// TwinCAT 3 PLC project M1L0_PLC
// ProgramVersion: 3.1.4020.5
// libraries:
//   Tc2_MC2, * (Beckhoff Automation GmbH)
//   Tc2_Standard, * (Beckhoff Automation GmbH)
//   Tc2_System, * (Beckhoff Automation GmbH)
//   Tc2_Utilities, * (Beckhoff Automation GmbH)
//   Tc3_Module, * (Beckhoff Automation GmbH)
//   lcls-twincat-motion,0.0.0,SLAC
// project tree:
//   / PlcTask.TcTTO
//   POUs/ MAIN.TcPOU
// real-time tasks:
//   TASK PlcTask: cycle T#10ms, priority 20, ADS port 350
// motion (NC):
//   TASK NC-Task 1 SAF: cycle T#2ms, priority 4, ADS port 501
//   TASK NC-Task 1 SVB: cycle T#10ms, priority 8, ADS port 511
//   AXIS Axis_Yup (id 1)
//     Dynamic: Acceleration=0.2, Deceleration=0.2, DelayTime=0.008
//     Velo: Maximum=0.45
//     OtherSettings: AllowMotionCmdToSlave=true
//     encoder EncType=1
//       EncPara: ScaleFactorNumerator=1e-006
//     drive DrvType=5
//       DrvPara: Inverse=true
//         Analog: VeloReferenz=0.48828125, ScaleFactorActTorque=0.1
//         TimeComp: TaskDelayCycles=1
//     controller CtrType=2
//       CtrPara: PriorControlFactor=1
//         PosDiffControl: Range=0.5
//         PID: PosKp=20, PosExtKp=5, DeadBandPosition=0.0004
//         Observer: BandWidth=20
//   AXIS Axis_Ydwn (id 2)
//     Dynamic: Acceleration=0.2, Deceleration=0.2, DelayTime=0.008
//     Velo: Maximum=0.45
//     OtherSettings: AllowMotionCmdToSlave=true
//     encoder EncType=1
//       EncPara: ScaleFactorNumerator=1e-006
//     drive DrvType=5
//       DrvPara: Inverse=true
//         Analog: VeloReferenz=0.48828125, ScaleFactorActTorque=0.1
//         TimeComp: TaskDelayCycles=1
//     controller CtrType=2
//       CtrPara: PriorControlFactor=1
//         PosDiffControl: Range=0.5
//         PID: PosKp=20, PosExtKp=5, DeadBandPosition=0.0004
//         Observer: BandWidth=20
//   AXIS Axis_Xup (id 3)
//     Dynamic: Acceleration=2, Deceleration=2, DelayTime=0.008
//     Velo: Maximum=1
//     OtherSettings: AllowMotionCmdToSlave=true
//     encoder EncType=1
//       EncPara: ScaleFactorNumerator=1e-006
//     drive DrvType=5
//       Analog: VeloReferenz=1.220703125, ScaleFactorActTorque=0.1
//       TimeComp: TaskDelayCycles=1
//     controller CtrType=2
//       CtrPara: PriorControlFactor=1
//         PosDiffControl: Range=0.1
//         PID: PosKp=10, PosExtKp=1, DeadBandPosition=0.0004
//         Observer: BandWidth=20
//   AXIS Axis_Xdwn (id 4)
//     Dynamic: Acceleration=2, Deceleration=2, DelayTime=0.008
//     Velo: Maximum=1
//     OtherSettings: AllowMotionCmdToSlave=true
//     encoder EncType=1
//       EncPara: ScaleFactorNumerator=1e-006
//     drive DrvType=5
//       DrvPara: Inverse=true
//         Analog: VeloReferenz=1.220703125, ScaleFactorActTorque=0.1
//         TimeComp: TaskDelayCycles=1
//     controller CtrType=2
//       CtrPara: PriorControlFactor=1
//         PosDiffControl: Range=0.1
//         PID: PosKp=10, PosExtKp=1, DeadBandPosition=0.0004
//         Observer: BandWidth=20
//   AXIS Axis_PitchCoarse (id 5)
//     General: UnitName=urad
//     Dynamic: Acceleration=390, Deceleration=390, DelayTime=0.008
//     Velo: Maximum=760
//     OtherSettings: AllowMotionCmdToSlave=true
//     encoder EncType=1
//       EncPara: ScaleFactorNumerator=0.001949317739
//     drive DrvType=5
//       Analog: VeloReferenz=761.4522417, ScaleFactorActTorque=0.1
//       TimeComp: TaskDelayCycles=1
//     controller CtrType=2
//       CtrPara: PriorControlFactor=1
//         PosDiffControl: Range=150
//         PID: PosKp=10, PosExtKp=1, DeadBandPosition=0.1
//         Observer: BandWidth=20
//   AXIS Axis_Bender (id 6)
//     Dynamic: Acceleration=0.1, Deceleration=0.1, DelayTime=0.008
//     Velo: Maximum=0.19
//     OtherSettings: AllowMotionCmdToSlave=true
//     encoder EncType=1
//       EncPara: ScaleFactorNumerator=1e-006
//     drive DrvType=5
//       Analog: VeloReferenz=0.1953125, ScaleFactorActTorque=0.1
//       TimeComp: TaskDelayCycles=1
//     controller CtrType=2
//       CtrPara: PriorControlFactor=1
//         PosDiffControl: Range=0.005
//         PID: PosKp=10, PosExtKp=1, DeadBandPosition=4e-005
//         Observer: BandWidth=20

CONFIGURATION M1L0_PLC
    RESOURCE PLC ON TwinCAT3
        TASK PlcTask(INTERVAL := T#10ms, PRIORITY := 20);
        PROGRAM MAIN WITH PlcTask : MAIN;
    END_RESOURCE
END_CONFIGURATION

// ---- POUs/MAIN.TcPOU
PROGRAM MAIN

VAR
//	{attribute 'TcLinkTo' := '.bLimFwd:=TIIB[y_up]^STM Status^Status^Digital input 1; .bLimBwd:=TIIB[y_up]^STM Status^Status^Digital input 2; .bSTO:=TIIB[di]^Channel 1^Input'}	
	{attribute 'TcLinkTo':='.bLimFwd:=TIIB[y_up]^STM Status^Status^Digital input 1'}		
    M1: DUT_MotionStage:=(nCommand:=3); // Yup
//	{attribute 'TcLinkTo' := '.bLimFwd:=TIIB[y_dwn]^STM Status^Status^Digital input 1; .bLimBwd:=TIIB[y_dwn]^STM Status^Status^Digital input 2'}
	M2: DUT_MotionStage:=(nCommand:=3); // Ydwn
//	{attribute 'TcLinkTo' := '.bLimFwd:=TIIB[x_up]^STM Status^Status^Digital input 1; .bLimBwd:=TIIB[x_up]^STM Status^Status^Digital input 2'}	
	M3: DUT_MotionStage:=(nCommand:=3); // Xup
//	{attribute 'TcLinkTo' := '.bLimFwd:=TIIB[x_dwn]^STM Status^Status^Digital input 1; .bLimBwd:=TIIB[x_dwn]^STM Status^Status^Digital input 2'}
	M4: DUT_MotionStage:=(nCommand:=3); // Xdwn
//	{attribute 'TcLinkTo' := '.bLimFwd:=TIIB[pitch]^STM Status^Status^Digital input 1; .bLimBwd:=TIIB[pitch]^STM Status^Status^Digital input 2'}	
	M5: DUT_MotionStage:=(nCommand:=3); // PitchCoarse
//	{attribute 'TcLinkTo' := '.bLimFwd:=TIIB[pitch]^STM Status^Status^Digital input 1; .bLimBwd:=TIIB[pitch]^STM Status^Status^Digital input 2'}	
	M6: DUT_MotionStage:=(nCommand:=3); // Bender
	fbMotionStage_x_up, fbMotionStage_x_dwn, fbMotionStage_y_up, fbMotionStage_y_dwn, fbMotionStage_pitch, fbMotionStage_bender : FB_MotionStage;
	stoEnable AT %I* : BOOL;
	{attribute 'TcLinkTo' := '.Count:=TIIB[1-x_up_2-x_dwn]^FB Inputs Channel 1^Position'}	
	x_up_enc  AT %I*: ST_RenishawAbsEnc;
	{attribute 'TcLinkTo' := '.Count:=TIIB[1-x_up_2-x_dwn]^FB Inputs Channel 2^Position'}
	x_dwn_enc  AT %I*: ST_RenishawAbsEnc;
	{attribute 'TcLinkTo' := '.Count:=TIIB[1-y_up_2-y_dwn]^FB Inputs Channel 1^Position'}	
	y_up_enc  AT %I*: ST_RenishawAbsEnc;
	{attribute 'TcLinkTo' := '.Count:=TIIB[1-y_up_2-y_dwn]^FB Inputs Channel 2^Position'}
	y_dwn_enc  AT %I*: ST_RenishawAbsEnc;
	// Auto coupling function block
	fbAutoCoupleX : FB_GantryAutoCoupling;
	fbAutoCoupleY : FB_GantryAutoCoupling;
	bExecuteCoupleX : BOOL;
	bExecuteCoupleY : BOOL;
	bExecuteDecoupleX : BOOL;
	bExecuteDecoupleY : BOOL;
	bGantryAlreadyCoupledX : BOOL;
	bGantryAlreadyCoupledY : BOOL;
	
	// Gantry variables
	nCurrGantryX : LINT;
	nCurrGantryY : LINT;
	nGantryTolX : LINT := 50000;
	nGantryTolY : LINT := 50000;
END_VAR

// Buttons to enable motors: write 0 to enable, 2 to disable
M1.nEnableMode; // Yup
M2.nEnableMode; // Ydwn
M3.nEnableMode; // Xup
M4.nEnableMode; // Xdwn
M5.nEnableMode; // PitchCoarse

// Encoder Reference Values: Starting motor positions prior to checkout
//y_up_enc.Ref := ;
//y_dwn_enc.Ref := ; Use initial motor positions for now
//x_up_enc.Ref := ; 
//x_dwn_enc.Ref := ;

// Gantry Differences to monitor
nCurrGantryY := ((ULINT_TO_LINT(y_up_enc.Count) - ULINT_TO_LINT(y_up_enc.Ref)) - (ULINT_TO_LINT(y_dwn_enc.Count) - ULINT_TO_LINT(y_dwn_enc.Ref)));
nCurrGantryX := ((ULINT_TO_LINT(x_up_enc.Count) - ULINT_TO_LINT(x_up_enc.Ref)) - (ULINT_TO_LINT(x_dwn_enc.Count) - ULINT_TO_LINT(x_dwn_enc.Ref)));

// E-stop
M1.bHardwareEnable := stoEnable;
M2.bHardwareEnable := stoEnable;
M3.bHardwareEnable := stoEnable;
M4.bHardwareEnable := stoEnable;
M5.bHardwareEnable := stoEnable;
M6.bHardwareEnable := stoEnable;


// Start Autocoupling
fbAutoCoupleX(nGantryTol:=nGantryTolX, Master:=M3, MasterEnc:=x_up_enc, Slave:=M4,
	          SlaveEnc:=x_dwn_enc, bExecuteCouple:=bExecuteCoupleX,
              bExecuteDecouple:=bExecuteDecoupleX,
              bGantryAlreadyCoupled=>bGantryAlreadyCoupledX);

fbAutoCoupleY(nGantryTol:=nGantryTolY, Master:=M1, MasterEnc:=y_up_enc, Slave:=M2,
	          SlaveEnc:=y_dwn_enc, bExecuteCouple:=bExecuteCoupleY,
              bExecuteDecouple:=bExecuteDecoupleY,
			  bGantryAlreadyCoupled=>bGantryAlreadyCoupledY);

fbMotionStage_y_up  (stMotionStage:=M1);
fbMotionStage_y_dwn (stMotionStage:=M2);
fbMotionStage_x_up  (stMotionStage:=M3);
fbMotionStage_x_dwn (stMotionStage:=M4);
fbMotionStage_pitch (stMotionStage:=M5);
fbMotionStage_bender (stMotionStage:=M6);

END_PROGRAM
